ABB RAPID module: TCP_mtip_tool2_nest_new.mod

MODULE TCP_mtip_tool2_nest_new
	! Points are read in order of declaration.
  ! Please do not change the order of points!

  LOCAL PERS robtarget pTCP_Point1:=[[920.7693,-672.4167,256.1491],[0.421933650970459,0.446557819843292,-0.785544514656067,0.0740130320191383],[-1,-3,1,1],[9E+09,9E+09,9E+09,9E+09,9E+09,9E+09]];
	LOCAL PERS robtarget pTCP_Point2:=[[937.9245,-887.7251,348.9297],[0.347764134407043,0.283149242401123,-0.893798351287842,0.00333250570110977],[-1,-3,1,1],[9E+09,9E+09,9E+09,9E+09,9E+09,9E+09]];
	LOCAL PERS robtarget pTCP_Point3:=[[844.739,-1250.37,396.9317],[0.215821132063866,0.227679237723351,-0.926976978778839,-0.205662533640862],[-1,-3,1,1],[9E+09,9E+09,9E+09,9E+09,9E+09,9E+09]];
	LOCAL PERS robtarget pTCP_Point4:=[[528.9692,-1565.36,309.8902],[0.0339936017990112,0.00803164020180702,-0.923155605792999,-0.382836282253265],[-1,-2,1,1],[9E+09,9E+09,9E+09,9E+09,9E+09,9E+09]];
	LOCAL PERS robtarget pTCP_Point5:=[[293.0721,-1431.188,388.4799],[0.0111524648964405,0.375994652509689,0.874071776866913,0.307412028312683],[-1,-2,1,1],[9E+09,9E+09,9E+09,9E+09,9E+09,9E+09]];
	LOCAL PERS robtarget pTCP_Point6:=[[234.4254,-1328.178,423.7864],[0.192174136638641,-0.118274301290512,0.957563877105713,0.179309040307999],[-1,-2,0,1],[9E+09,9E+09,9E+09,9E+09,9E+09,9E+09]];
	LOCAL PERS robtarget pTCP_Point7:=[[335.6236,-1028.312,511.4952],[0.088929682970047,-0.274992287158966,0.956745743751526,-0.0332922786474228],[-1,-2,0,1],[9E+09,9E+09,9E+09,9E+09,9E+09,9E+09]];
	LOCAL PERS robtarget pTCP_Point8:=[[440.8602,-859.3893,502.0867],[0.0406301915645599,0.490927517414093,-0.862156629562378,0.118428446352482],[-1,-3,0,1],[9E+09,9E+09,9E+09,9E+09,9E+09,9E+09]];

ENDMODULE
